{attribute 'pack_mode' := '2'}
TYPE ST_LIST_STATE :
STRUCT
  Init        : E_PROGRESS;
  State       : E_LIST_STATE;

  Free        : UDINT;
  Count       : UDINT;
END_STRUCT
END_TYPE

(* stored: Version 1.1.0.1
   DUT ST_LIST_STATE: Id {f63745ba-b45f-42fc-87ce-b953caf56c67} *)
